//   NC SAF/Axes/Mover Axis 3 <-> TcCOM Objects/XtsProcessingUnit 1/Mover 3
//     SoftDrive 3/Data Pointer/InputPointer1 <-> Inputs/SoftDriveInput
//     SoftDrive 3/Data Pointer/OutputPointer1 <-> Outputs/SoftDriveOutput
//   NC SAF/Axes/Mover Axis 4 <-> TcCOM Objects/XtsProcessingUnit 1/Mover 4
//     SoftDrive 4/Data Pointer/InputPointer1 <-> Inputs/SoftDriveInput
//     SoftDrive 4/Data Pointer/OutputPointer1 <-> Outputs/SoftDriveOutput
//   NC SAF/Axes/Mover Axis 5 <-> TcCOM Objects/XtsProcessingUnit 1/Mover 5
//     SoftDrive 5/Data Pointer/InputPointer1 <-> Inputs/SoftDriveInput
//     SoftDrive 5/Data Pointer/OutputPointer1 <-> Outputs/SoftDriveOutput
//   NC SAF/Axes/Mover Axis 6 <-> TcCOM Objects/XtsProcessingUnit 1/Mover 6
//     SoftDrive 6/Data Pointer/InputPointer1 <-> Inputs/SoftDriveInput
//     SoftDrive 6/Data Pointer/OutputPointer1 <-> Outputs/SoftDriveOutput
//   NC SAF/Axes/Mover Axis 7 <-> TcCOM Objects/XtsProcessingUnit 1/Mover 7
//     SoftDrive 7/Data Pointer/InputPointer1 <-> Inputs/SoftDriveInput
//     SoftDrive 7/Data Pointer/OutputPointer1 <-> Outputs/SoftDriveOutput
//   NC SAF/Axes/Mover Axis 8 <-> TcCOM Objects/XtsProcessingUnit 1/Mover 8
//     SoftDrive 8/Data Pointer/InputPointer1 <-> Inputs/SoftDriveInput
//     SoftDrive 8/Data Pointer/OutputPointer1 <-> Outputs/SoftDriveOutput
//   NC SAF/Axes/Mover Axis 9 <-> TcCOM Objects/XtsProcessingUnit 1/Mover 9
//     SoftDrive 9/Data Pointer/InputPointer1 <-> Inputs/SoftDriveInput
//     SoftDrive 9/Data Pointer/OutputPointer1 <-> Outputs/SoftDriveOutput
//   Main Instance <-> NC SAF/Axes/Mover Axis 1
//     PlcTask Inputs/MAIN.Mover[0].AxisReference.NcToPlc <-> Outputs/ToPlc
//     PlcTask Outputs/MAIN.Mover[0].AxisReference.PlcToNc <-> Inputs/FromPlc
//   Main Instance <-> NC SAF/Axes/Mover Axis 10
//     PlcTask Inputs/MAIN.Mover[9].AxisReference.NcToPlc <-> Outputs/ToPlc
//     PlcTask Outputs/MAIN.Mover[9].AxisReference.PlcToNc <-> Inputs/FromPlc
//   Main Instance <-> NC SAF/Axes/Mover Axis 2
//     PlcTask Inputs/MAIN.Mover[1].AxisReference.NcToPlc <-> Outputs/ToPlc
//     PlcTask Outputs/MAIN.Mover[1].AxisReference.PlcToNc <-> Inputs/FromPlc
//   Main Instance <-> NC SAF/Axes/Mover Axis 3
//     PlcTask Inputs/MAIN.Mover[2].AxisReference.NcToPlc <-> Outputs/ToPlc
//     PlcTask Outputs/MAIN.Mover[2].AxisReference.PlcToNc <-> Inputs/FromPlc
//   Main Instance <-> NC SAF/Axes/Mover Axis 4
//     PlcTask Inputs/MAIN.Mover[3].AxisReference.NcToPlc <-> Outputs/ToPlc
//     PlcTask Outputs/MAIN.Mover[3].AxisReference.PlcToNc <-> Inputs/FromPlc
//   Main Instance <-> NC SAF/Axes/Mover Axis 5
//     PlcTask Inputs/MAIN.Mover[4].AxisReference.NcToPlc <-> Outputs/ToPlc
//     PlcTask Outputs/MAIN.Mover[4].AxisReference.PlcToNc <-> Inputs/FromPlc
//   Main Instance <-> NC SAF/Axes/Mover Axis 6
//     PlcTask Inputs/MAIN.Mover[5].AxisReference.NcToPlc <-> Outputs/ToPlc
//     PlcTask Outputs/MAIN.Mover[5].AxisReference.PlcToNc <-> Inputs/FromPlc
//   Main Instance <-> NC SAF/Axes/Mover Axis 7
//     PlcTask Inputs/MAIN.Mover[6].AxisReference.NcToPlc <-> Outputs/ToPlc
//     PlcTask Outputs/MAIN.Mover[6].AxisReference.PlcToNc <-> Inputs/FromPlc
//   Main Instance <-> NC SAF/Axes/Mover Axis 8
//     PlcTask Inputs/MAIN.Mover[7].AxisReference.NcToPlc <-> Outputs/ToPlc
//     PlcTask Outputs/MAIN.Mover[7].AxisReference.PlcToNc <-> Inputs/FromPlc
//   Main Instance <-> NC SAF/Axes/Mover Axis 9
//     PlcTask Inputs/MAIN.Mover[8].AxisReference.NcToPlc <-> Outputs/ToPlc
//     PlcTask Outputs/MAIN.Mover[8].AxisReference.PlcToNc <-> Inputs/FromPlc
//   Main Instance <-> NC SAF/Objects/Collision Avoidance
//     PlcTask Inputs/MAIN.GroupRef.NcToPlc <-> Group Outputs/ToPLC
//     PlcTask Outputs/MAIN.GroupRef.PlcToNc <-> Group Inputs/FromPLC

// ---- DUTs/HMI/HMIXTSHelper_typ.TcDUT
TYPE HMIXTSHelper_typ :
STRUCT
	Mover	: ARRAY[0..GVL.NUM_MOVERS-1] OF HMIXTSMoverHelper_typ;
END_STRUCT
END_TYPE

// ---- DUTs/HMI/HMIXTSMoverHelper_typ.TcDUT
TYPE HMIXTSMoverHelper_typ :
STRUCT
	BallImgVisibility:			BOOL;
	BallRejectImgVisibility:	BOOL;
	MoverTextVisibility: 		BOOL;
	MoverText: 					STRING;
END_STRUCT
END_TYPE

// ---- DUTs/IO/BallSeat/BallSeat_Inputs_typ.TcDUT
TYPE BallSeat_Inputs_typ:
STRUCT
	BallClampOpened AT %I*: BOOL;
	BallClampClosed AT %I*: BOOL;
	BallSeatExtended AT %I*: BOOL;
	BallSeatRetracted AT %I*: BOOL;
END_STRUCT
END_TYPE

// ---- DUTs/IO/BallSeat/BallSeat_Outputs_typ.TcDUT
TYPE BallSeat_Outputs_typ:
STRUCT
	BallClampOpen AT %Q*: BOOL;
	BallClampClose AT %Q*: BOOL;
	ExtendBallSeater AT %Q*: BOOL;
	RetractBallSeater AT %Q*: BOOL;
END_STRUCT
END_TYPE

// ---- DUTs/IO/Orient/Orient_IO_typ.TcDUT
TYPE Orient_IO_typ:
STRUCT
	Inputs	: Orient_Inputs_typ;
	Outputs	: Orient_Outputs_typ;
END_STRUCT
END_TYPE

// ---- DUTs/IO/Orient/Orient_Outputs_typ.TcDUT
TYPE Orient_Outputs_typ:
STRUCT
	BallClampOpen AT %Q*: BOOL;
	BallClampClose AT %Q*: BOOL;
	LoadBall AT %Q*: BOOL;
END_STRUCT
END_TYPE

// ---- DUTs/IO/IO_typ.TcDUT
TYPE IO_typ:
STRUCT
	Orient: 	Orient_IO_typ;
	BallSeat:	BallSeat_IO_typ;
	Print:		Print_IO_typ;
	Vision:		Vision_IO_typ;
	Kickout:	Kickout_IO_typ;
	TrayLoad:	TrayLoad_IO_typ;
END_STRUCT
END_TYPE

// ---- DUTs/IO/Print/Print_Inputs_typ.TcDUT
TYPE Print_Inputs_typ:
STRUCT
	PrintActive AT %I*: BOOL;
	PrintComplete AT %I*: BOOL;
END_STRUCT
END_TYPE

// ---- DUTs/IO/Print/Print_IO_typ.TcDUT
TYPE Print_IO_typ:
STRUCT
	Inputs	: Print_Inputs_typ;
	Outputs	: Print_Outputs_typ;
END_STRUCT
END_TYPE

// ---- DUTs/IO/Print/Print_Outputs_typ.TcDUT
TYPE Print_Outputs_typ:
STRUCT
	Print AT %Q*: BOOL;
END_STRUCT
END_TYPE

// ---- DUTs/IO/TrayLoad/TrayLoad_Inputs_typ.TcDUT
TYPE TrayLoad_Inputs_typ:
STRUCT
	BallClampOpened AT %I*: BOOL;
	BallClampClosed AT %I*: BOOL;
	TrayLoadComplete AT %I*: BOOL;
END_STRUCT
END_TYPE

// ---- DUTs/IO/TrayLoad/TrayLoad_IO_typ.TcDUT
TYPE TrayLoad_IO_typ:
STRUCT
	Inputs	: TrayLoad_Inputs_typ;
	Outputs	: TrayLoad_Outputs_typ;
END_STRUCT
END_TYPE

// ---- DUTs/IO/TrayLoad/TrayLoad_Outputs_typ.TcDUT
TYPE TrayLoad_Outputs_typ:
STRUCT
	BallClampOpen AT %Q*: BOOL;
	BallClampClose AT %Q*: BOOL;
	LoadTray AT %Q*: BOOL;
END_STRUCT
END_TYPE

// ---- DUTs/IO/Vision/Vision_Inputs_typ.TcDUT
TYPE Vision_Inputs_typ:
STRUCT
	VisionActive AT %I*: BOOL;
	VisionPass AT %I*: BOOL;
	VisionFail AT %I*: BOOL;
END_STRUCT
END_TYPE

// ---- DUTs/IO/Vision/Vision_IO_typ.TcDUT
TYPE Vision_IO_typ:
STRUCT
	Inputs	: Vision_Inputs_typ;
	Outputs	: Vision_Outputs_typ;
END_STRUCT
END_TYPE

// ---- POUs/XTS/BallPrinterStations/DUT/PrintConfig_typ.TcDUT
TYPE PrintConfig_typ :
STRUCT
	StationEnable	: ARRAY[0..GVL.MULTISTN_NUM_STN - 1] OF BOOL;
	ProcessIndex	: ARRAY[0..GVL.MULTISTN_NUM_STN - 1] OF USINT;
	FinalPrint		: ARRAY[0..GVL.MULTISTN_NUM_STN - 1] OF BOOL;
	LastProcessIndex0StnIndex	: USINT;
END_STRUCT
END_TYPE

// ---- POUs/XTS/BallPrinterStations/DUT/StnState_Enum.TcDUT
(*{attribute 'qualified_only'}*)
{attribute 'strict'}
TYPE StnState_Enum :
(
	STN_WAIT				:= 0,
	STN_CHECKMOVER			:= 1,
	STN_OPENBALLCLAMP		:= 2,
	STN_PROCESS				:= 3,
	STN_CLOSEBALLCLAMP		:= 4,
	STN_SEND				:= 5,
	STN_ERROR				:= 10
);
END_TYPE

// ---- GVLs/GVL.TcGVL
{attribute 'qualified_only'}
VAR_GLOBAL CONSTANT

    NUM_MOVERS   		: USINT := 10;   	// This should be set to the exact number of movers on the system
	NUM_ZONES			: USINT := 1;
    NUM_STATIONS 		: USINT := 5;   	// This should be set to a value equal to or greater than the number of stations needed
    NUM_MULTISTATIONS 	: USINT := 2;   	// This should be set to a value equal to or greater than the number of Multi stations needed
	MULTISTN_NUM_STN	: USINT := 4;		// This should be set to a value equal to or greater than the max number of stations in a multi station

    TRACK_LENGTH 		: LREAL := 3000;	// This should be set to the exact length [mm] of the track system

	STN_ORIENT		: USINT := 0;
	STN_BALLSEAT	: USINT := 1;
	STN_VISION		: USINT := 2;
	STN_KICKOUT		: USINT := 3;

	MULTISTN_PRINT		: USINT := 0;
	MULTISTN_TRAYLOAD	: USINT := 1;

    {attribute 'TcInitSymbol'}
    pXtsProcessingUnit : OTCID:=0; // This pointer needs to be initialized in the Main Instance, under Symbol Initialization

	NUM_TRACKS  : USINT := 1;	// This is the number of logical tracks in the system

END_VAR
VAR_GLOBAL
	newCallTime: LREAL;
END_VAR

// ---- ITFs/iMover.TcIO
INTERFACE iMover

METHOD ActivateTrack : BOOL
VAR_INPUT
	Track	: REFERENCE TO Track;
END_VAR
END_METHOD

{attribute 'monitoring' := 'call'}
PROPERTY CurrentDestinationPosition : LREAL
GET
END_GET
END_PROPERTY

{attribute 'monitoring' := 'call'}
PROPERTY CurrentMoveType : MoverCommandType_enum
GET
END_GET
END_PROPERTY

PROPERTY CurrentObjective : String
GET
END_GET
END_PROPERTY

PROPERTY CurrentTrack : POINTER TO Track
GET
END_GET
END_PROPERTY

METHOD Cyclic : iMover
VAR_IN_OUT
	GroupReference		: AXES_GROUP_REF;
END_VAR
END_METHOD

METHOD CyclicTrack : BOOL
VAR
END_VAR
END_METHOD

METHOD Disable : iMover
VAR_INPUT
END_VAR
END_METHOD

METHOD Enable : iMover
VAR_INPUT
END_VAR
END_METHOD

METHOD GroupStop : iMover
VAR_INPUT
END_VAR
END_METHOD

METHOD Halt : iMover
VAR_INPUT
END_VAR
END_METHOD

PROPERTY IsTrackReady : BOOL
GET
END_GET
END_PROPERTY

METHOD LogUserEvent : iMover
VAR_INPUT
	String1	: STRING;	// First content section of user-event message
	String2 : STRING;	// Second content section of user-event message
	String3 : STRING;	// Third content section of user-event message
END_VAR
END_METHOD

METHOD PUBLIC MoveToPosition : iMover
VAR_INPUT
	
	DestinationPosition		: LREAL;	// position on track for a shuttle to move towards

END_VAR
END_METHOD

METHOD MoveToStation : iMover
VAR_INPUT
	DestinationStation	: REFERENCE TO Station;	
END_VAR
END_METHOD

METHOD MoveVelocity : iMover
VAR_INPUT
	DesiredVelocity : LREAL;		//The velocity to be commanded [mm/s]
END_VAR
END_METHOD

PROPERTY Payload : Payload_typ
GET
END_GET
SET
END_SET
END_PROPERTY

METHOD ReissueCommand : iMover
VAR_INPUT
END_VAR
END_METHOD


METHOD SetAcceleration : iMover
VAR_INPUT
	Acceleration	: LREAL;
END_VAR
END_METHOD

METHOD SetDeceleration : iMover
VAR_INPUT
	Deceleration	: LREAL;
END_VAR
END_METHOD

METHOD SetDirection : iMover
VAR_INPUT
	Direction		: Tc3_Mc3Definitions.MC_Direction;
END_VAR
END_METHOD

METHOD SetJerk : iMover
VAR_INPUT
	Jerk		: LREAL;
END_VAR
END_METHOD

METHOD SetVelocity : iMover
VAR_INPUT
	Velocity		: LREAL;		// Updates Mover's internal velocity parameter. Takes effect immediately. [mm/s]
END_VAR
END_METHOD

METHOD SyncToAxis : iMover
VAR_INPUT
	
	MasterAxis		: REFERENCE TO AXIS_REF;
	MasterSyncPos	: LREAL;	// Master sync position (nonmodulo), where the input axis will be located when first synchronized
	SlaveSyncPos	: LREAL;	// Mover sync position, where the mover will be located when first synchronized
	SyncStrategy	: MC_SYNC_STRATEGY;	// Direction input
	
END_VAR
END_METHOD

METHOD SyncToMover : iMover
VAR_INPUT

	MasterMover		: REFERENCE TO Mover;	// Synchronization master mover, whose position to follow. Further motion commands break the pairing
	Gap				: LREAL;				// Gap distance to lead mover. Positive values indicate following, negative values indicate leading

END_VAR
END_METHOD

END_INTERFACE

// ---- POUs/XTS/Station.TcPOU
FUNCTION_BLOCK Station EXTENDS Objective
VAR

    {attribute 'hide'}
    internalPosition : LREAL;
	internalTrackId : DINT := 1;

END_VAR

{attribute 'monitoring' := 'variable'}
PROPERTY CurrentMover : REFERENCE TO Mover
GET
VAR

    i          : ULINT;
    difference : LREAL;

	moverTrackId: INT;
END_VAR
// default to unassigned
CurrentMover REF= 0;

FOR i := 0 TO SIZEOF(internalTrackedMovers) / SIZEOF(internalTrackedMovers[0]) - 1 DO

    // In order to deal with the rollover, we need to evaluate distance between congruence classes
    // e.g. On a 4m track, if the Station is at 0.34mm and the Mover is at 3999.8mm, then this is considered 'in position'	

    IF internalTrackedMovers[i] <> 0 THEN
		moverTrackId := internalTrackedMovers[i]^.CurrentTrack^.Id;
		IF (moverTrackId = internalTrackId) THEN

			difference := Position - internalTrackedMovers[i]^.TrackInfo.TrackPosition;
			// un-wrap if necessary
			IF (difference < 0) THEN 
				difference := difference + GVL.TRACK_LENGTH;
			END_IF
	
			IF (difference < 1.0) AND NOT internalTrackedMovers[i]^.Busy THEN
				CurrentMover                    REF= internalTrackedMovers[i]^;
				CurrentMover.SourceInstancePath := THIS^.InstancePath;
				// Exit;	// CW - shouldn't this be here?
			END_IF
		END_IF
    END_IF

END_FOR

// If the Station has no CurrentMover, then return an imposter ErrorMover, whose method calls all trigger an error message
IF __ISVALIDREF(CurrentMover) = FALSE THEN
    ErrorMover.SourceInstancePath := THIS^.InstancePath;
    CurrentMover                  REF= ErrorMover;
END_IF
END_GET
END_PROPERTY

METHOD Cyclic : BOOL

VAR
    i : USINT;
END_VAR
FOR i := 0 TO GVL.NUM_MOVERS - 1 DO

    // This mover is no longer destined for any station
    IF internalTrackedMovers[i] <> 0 AND_THEN internalTrackedMovers[i]^.CurrentMoveType <> MOVETYPE_STATION THEN
        internalTrackedMovers[i] := 0;
        // This mover is no longer destined for this specific station. Comparing instance path seems to be the best way to do this comparison?
    ELSIF internalTrackedMovers[i] <> 0 AND_THEN internalTrackedMovers[i]^.CurrentObjective <> InstancePath THEN
        internalTrackedMovers[i] := 0;
    END_IF

END_FOR
END_METHOD

{attribute 'monitoring' := 'variable'}
PROPERTY MoverInPosition : BOOL
GET
VAR

    i          : ULINT;
    difference : LREAL;
	moverTrackId: INT;
END_VAR
// default to false
MoverInPosition := FALSE;

FOR i := 0 TO SIZEOF(internalTrackedMovers) / SIZEOF(internalTrackedMovers[0]) - 1 DO

    // In order to deal with the rollover, we need to evaluate distance between congruence classes
    // e.g. On a 4m track, if the Station is at 0.34 mm and the Mover is at 3999.8mm, then this is considered 'in position' 

    // todo: make in-position tolerance adjustable. add condition that mover is stopped?
    IF internalTrackedMovers[i] <> 0 THEN
		moverTrackId := internalTrackedMovers[i]^.CurrentTrack^.Id;
		IF (moverTrackId = internalTrackId) THEN
			difference := Position - internalTrackedMovers[i]^.TrackInfo.TrackPosition;
			// un-wrap if necessary
			IF (difference < 0) THEN 
				difference := difference + GVL.TRACK_LENGTH;
			END_IF

			IF (difference < 1.0) AND NOT internalTrackedMovers[i]^.Busy THEN
				MoverInPosition := TRUE;
			END_IF
		END_IF;
    END_IF;

END_FOR
END_GET
END_PROPERTY

{attribute 'monitoring' := 'call'}
PROPERTY Position : LREAL
GET
Position := internalPosition;
END_GET
SET
internalPosition := Position;
END_SET
END_PROPERTY

PROPERTY TrackId : DINT
GET
TrackId := internalTrackId;
END_GET
SET
internalTrackId := TrackId;
END_SET
END_PROPERTY

END_FUNCTION_BLOCK

// ---- POUs/XTS/Objective.TcPOU
{attribute 'reflection'}
(*{attribute 'hide_all_locals'}*)
FUNCTION_BLOCK ABSTRACT Objective
VAR_INPUT
END_VAR
VAR

    internalTrackedMoverCount 	: USINT;
   
    internalTrackedMovers 		: ARRAY[0..GVL.NUM_MOVERS - 1] OF POINTER TO Mover;

    ErrorMover 					: ErrorMover;
	
    {attribute 'instance-path'}
    {attribute 'noinit'}
    InstancePath 				: STRING; // Unique variable path of the instance	
END_VAR
VAR_OUTPUT
END_VAR

PROPERTY CurrentMover : Reference to Mover
GET

// If no real mover can be returned as Current, return an imposter instead to output error messages
IF __ISVALIDREF( CurrentMover ) = FALSE THEN
	ErrorMover.SourceInstancePath	:= THIS^.InstancePath;
	CurrentMover					REF= ErrorMover;
END_IF
END_GET
END_PROPERTY

METHOD RegisterMover : BOOL
VAR_INPUT
    NewMover : REFERENCE TO Mover;
END_VAR

VAR
    i              : ULINT;
    duplicateFound : BOOL;
    emptyIDX       : ulint;
END_VAR
(*
	Add a mover to a list of movers tracked by the objective.
	Movers can't be added multiple times, so check for duplicates
	Movers can't overwrite others in the list, so check that the array element is clear
*)

IF __ISVALIDREF(NewMover) THEN // validate reference

    duplicateFound            := FALSE; // default to false, counterexample below
    internalTrackedMoverCount := 0;     // reset to zero, incremented below

    FOR i := 0 TO SIZEOF(internalTrackedMovers) / SIZEOF(internalTrackedMovers[i]) - 1 DO
        IF internalTrackedMovers[i] <> 0 THEN
            IF ADR(NewMover) = internalTrackedMovers[i] THEN
                duplicateFound := TRUE; // this mover already tracked
            END_IF

            internalTrackedMoverCount := internalTrackedMoverCount + 1;
        ELSE
            emptyIDX := i; // confirmed open array element
        END_IF
    END_FOR

    IF duplicateFound = FALSE THEN
        internalTrackedMovers[emptyIDX] := ADR(NewMover); // new mover goes into open array element
        internalTrackedMoverCount       := internalTrackedMoverCount + 1;
    END_IF

ELSE
    ADSLOGSTR(ADSLOG_MSGTYPE_LOG, 'Error: Mover input is invalid', '');
END_IF
END_METHOD

METHOD RegisterMoverList : BOOL
VAR_INPUT
    NewMoverList : iMoverList;
END_VAR
VAR
    i                : ULINT;
    duplicateFound   : BOOL;
    emptyIDX         : USINT;
    arrTrackedMovers : ARRAY[0..GVL.NUM_MOVERS - 1] OF POINTER TO Mover;
END_VAR
(*
	Adds an entire MoverList to the Tracked Movers of the objective.
*)

arrTrackedMovers := NewMoverList.TrackedMovers;

// IF __ISVALIDREF( NewMoverList ) THEN
IF NewMoverList <> 0 THEN
    FOR i := 0 TO SIZEOF(arrTrackedMovers) / SIZEOF(arrTrackedMovers[0]) - 1 DO

        THIS^.RegisterMover(arrTrackedMovers[i]^);

    END_FOR
END_IF
END_METHOD

{attribute 'monitoring' := 'call'}
PROPERTY TrackedMoverCount : USINT
GET
VAR
    i : INT;
END_VAR
TrackedMoverCount := 0;

FOR i := 0 TO GVL.NUM_MOVERS - 1 DO

    IF internalTrackedMovers[i] <> 0 THEN
        TrackedMoverCount := TrackedMoverCount + 1;
    END_IF

END_FOR
END_GET
END_PROPERTY

PROPERTY TrackedMovers : ARRAY[0..GVL.NUM_MOVERS - 1] OF POINTER TO Mover
GET
TrackedMovers := internalTrackedMovers;
END_GET
END_PROPERTY

METHOD UnregisterAll : BOOL
VAR_INPUT
END_VAR
VAR
    i : USINT;
END_VAR
// Blow out the tracked mover array
memset(ADR(internalTrackedMovers), 0, SIZEOF(internalTrackedMovers));
END_METHOD

METHOD UnregisterCurrent : BOOL
VAR_INPUT
END_VAR
THIS^.UnregisterMover(CurrentMover);
END_METHOD

METHOD UnregisterMover : BOOL
VAR_INPUT
    RemovingMover : REFERENCE TO Mover;
END_VAR
VAR
    i              : dint;
    duplicateFound : BOOL;
END_VAR
(*
	Remove a mover to a list of movers tracked by the objective.
	Only movers in the list can be removed, otherwise nothing happens
*)

//	IF RemovingMover <> 0 THEN			// validate pointer
IF __ISVALIDREF(RemovingMover) THEN

    internalTrackedMoverCount := 0;

    FOR i := 0 TO SIZEOF(internalTrackedMovers) / SIZEOF(internalTrackedMovers[0]) - 1 DO
        IF internalTrackedMovers[i] <> 0 THEN // validate pointer

            internalTrackedMoverCount := internalTrackedMoverCount + 1;

            IF ADR(RemovingMover) = internalTrackedMovers[i] THEN
                internalTrackedMovers[i]  := 0; // remove the pointer
                internalTrackedMoverCount := internalTrackedMoverCount - 1;
            END_IF

        END_IF
    END_FOR

ELSE
    ADSLOGSTR(ADSLOG_MSGTYPE_LOG, 'Error: Mover input is invalid', '');
END_IF
END_METHOD

END_FUNCTION_BLOCK

// ---- POUs/MAIN.TcPOU
PROGRAM MAIN
VAR
	// Machine Stations
	OrientStation:		OrientStation;
	BallSeatStation:	BallSeatStation;
	PrintStation:		PrintStation;
	VisionStation:		VisionStation;
	SimTimers:			SimTimers_typ;

	// ========= System Control / FSM Variables =========
	
	MainCommands 		: MainCommands_typ; 	// command struct for cycling thru the state machine
	MainState    		: MainState_enum;   	// enumeration for the Main state machine

	// ========= Linked NC Variables & References =========
	
	Mover    			: ARRAY[0..GVL.NUM_MOVERS - 1] OF Mover; 	// instantiation of Mover objects. Matches the number of movers on the system
    GroupRef 			: AXES_GROUP_REF;                       	 // linked to the Collision Avoidance group and passed cyclically to every Mover object

	// ========= Objectives & Parameters =========

    MoverList    		: MoverList;
    ParameterSet 		: MotionParameters_typ;

    Station         	: ARRAY[0..GVL.NUM_STATIONS - 1] OF Station;
	MultiStation		: ARRAY[0..GVL.NUM_MULTISTATIONS - 1] OF MultiStation;
    Zone            	: ARRAY[0..0] OF Zone;

    // ========= Example Application Variables =========

    lowVelocity    		: LREAL := 200;  	// mm/s
    mediumVelocity 		: LREAL := 800;  	// mm/s
    highVelocity   		: LREAL := 1200; 	// mm/s

    // ========= Helper, State, & Index Variables =========
	
    i                	: UINT; 	// index variable; gets reused in various FOR loops
	j					: UINT;		// index variable; gets reused in various FOR loops
    n                	: UINT; 	// secondary index variable, for enabling movers
    allMoversEnabled 	: BOOL; 	// helper flag for verifying enable status of all movers
	allMoverTracksEnabled : BOOL;	// helper flag for verifying track active status of all movers
	allMoversDisabled	: BOOL;		// helper flag for verifying disable status of all movers
	allMoversHalted		: BOOL;		// helper flag for verifying halt status of all movers

    StationTimer 		: ARRAY[0..GVL.NUM_STATIONS-1] OF TON; // timer blocks, for station dwells	
    MultiStationTimer 	: ARRAY[0..GVL.NUM_MultiSTATIONS-1] OF TON; // timer blocks, for station dwells	
	
	// ========= XTS Utility Diagnostics =========
	
	VisuDiag						: FB_VisuXtsDiag;
	fbXtsEnvironment				: FB_TcIoXtsEnvironment;
	fbXtsEnvironmentVisu			: FB_XtsEnvironmentVisu;
	stXtsEnvironmentConfiguration	: ST_XtsEnvironmentConfiguration;
	nEnvironmentState				: INT;
	
	// ======== Track management ========
	Track		: ARRAY [0..GVL.NUM_TRACKS] OF Track;

	// IO
	IO: IO_typ;

	Payload: Payload_typ;
	HMIXTSHelper : HMIXTSHelper_typ;
END_VAR

(* ======================================================================================

--- XTS Starter Project ---

This MAIN (PRG) is intended to serve as an example, which can be modified to suit your specific application.

No programming changes should be necessary inside the provided XTS objects / function block definitions.
They are intended to be simply instantiated and controlled via the provided methods and properties.
However the objects are provided as open-source for modification and extension as needed.

Documentation for these objects can be found online at:
https://beckhoff-usa-community.github.io/XTS_Base/

Bug reports, new feature requests, and general feedback is always welcome on our Github page.
For any other questions, please reach out to your local Application Engineer.

- Beckhoff USA Advanced Applications Group

====================================================================================== *)
_AppInfo.KeepOutputsOnBP := TRUE;
CASE MainState OF
    MS_DISABLED: // --------------------------------------------------------- IDLE STATE
		(*Wait here until an operator issues a MainCommand to Enable the system. 
		Disallow Start and Stop commands until the system has been Enabled*)

        MainCommands.Start		:= FALSE;
		MainCommands.Stop		:= FALSE;
		
        IF MainCommands.Enable THEN
            MainCommands.Disable := FALSE;
            MainState            := MS_INITIALIZING_MOVERS;
        END_IF

    MS_INITIALIZING_MOVERS: // --------------------------------------------- SET MOVER MOTION PARAMETERS
		(*Initialize Mover motion parameters via a Parameter Set. Once complete, step
		forward to begin Enabling movers on the system*)
		
		ParameterSet.Jerk         := 1E5; // mm/s3
		ParameterSet.Acceleration := 1E4; // mm/s2
		ParameterSet.Deceleration := 1E4; // mm/s2
		ParameterSet.Velocity     := 1E3; // mm/s
		ParameterSet.Direction    := mcDirectionPositive;

        FOR i := 0 TO GVL.NUM_MOVERS - 1 DO
            Mover[i].MotionParameters := ParameterSet;
        END_FOR
		
		IF MainCommands.Disable THEN
			MainCommands.Enable		:= FALSE;
			MainState				:= MS_DISABLED;
		ELSIF MainCommands.Stop THEN
			MainCommands.Stop		:= FALSE;
			MainCommands.Disable	:= TRUE;
			MainCommands.Start		:= FALSE;
			MainState				:= MS_DISABLED;
		ELSIF MainCommands.Enable THEN
        	MainState 				:= MS_ONESHOT_ENABLE;
		END_IF

	MS_ONESHOT_ENABLE:	// -------------------------------------------------- SINGLE-CYCLE ISSUE ENABLE COMMANDS
		(*Begin Enabling movers by calling Mover.Enable(). Methods in this project
		are intended to be called once, although they will function correctly if called repeatedly*)

		FOR i := 0 TO GVL.NUM_MOVERS - 1 DO
			Mover[i].Enable();
		END_FOR

		MainState		:= MS_ENABLING_MOVERS;
	
    MS_ENABLING_MOVERS: // -------------------------------------------------- RESETTING AND ENABLING AXES
		(*Wait here until all movers have Enabled. This means that the Axis has
		fully energized, and also that all Collision Avoidance grouping and Mover 1 detection
		has finished. If the state machine gets stuck in this state, check the Error output
		of an individual Mover to see what the issue is. A common cause is forgetting to link
		Mover NC Axes to the AXIS_REF inside the PLC*)

        allMoversEnabled := TRUE; // default ...

        FOR i := 0 TO GVL.NUM_MOVERS - 1 DO
            IF Mover[i].Ready = FALSE THEN
                allMoversEnabled 		:= FALSE;
            END_IF
        END_FOR

        IF allMoversEnabled THEN
			IF MainCommands.Disable THEN
				MainCommands.Enable		:=FALSE;
            	MainState				:= MS_ONESHOT_DISABLE;
			ELSIF MainCommands.Stop	 THEN
				MainCommands.Start		:=FALSE;
				MainState				:= MS_ONESHOT_STOP;
			ELSIF MainCommands.Enable THEN
	        	MainState 				:= MS_INITIALIZING_OBJECTIVES;
			END_IF
        END_IF

    MS_INITIALIZING_OBJECTIVES: // --------------------------------------------- WRITING OBJECTIVE PARAMETERS
		(*Initialize Station positions, Position Trigger positions, Zones etc. *)

        // Initialize station positions
        Station[GVL.STN_ORIENT].Position	:= 800;
        Station[GVL.STN_BALLSEAT].Position	:= 900;
        Station[GVL.STN_VISION].Position	:= 2125;
        Station[GVL.STN_KICKOUT].Position	:= 2375;

		MultiStation[GVL.MULTISTN_PRINT].PositionTrigger.Position	:= 1541;
		MultiStation[GVL.MULTISTN_PRINT].Station[0].Position		:= 1621;
		MultiStation[GVL.MULTISTN_PRINT].Station[1].Position		:= 1707;
		MultiStation[GVL.MULTISTN_PRINT].Station[2].Position		:= 1793;
		MultiStation[GVL.MULTISTN_PRINT].Station[3].Position		:= 1879;

		MultiStation[GVL.MULTISTN_TRAYLOAD].PositionTrigger.Position	:= 41;
		MultiStation[GVL.MULTISTN_TRAYLOAD].Station[0].Position			:= 121;
		MultiStation[GVL.MULTISTN_TRAYLOAD].Station[1].Position			:= 207;
		MultiStation[GVL.MULTISTN_TRAYLOAD].Station[2].Position			:= 293;
		MultiStation[GVL.MULTISTN_TRAYLOAD].Station[3].Position			:= 379;

        Zone[0].StartPosition := 0;
        Zone[0].EndPosition   := 3000;

		// give all tracks their ID number
		FOR i := 0 TO GVL.NUM_TRACKS DO
			Track[i].Id := UINT_TO_INT(i);
		END_FOR
		
		// If a single logical track is used (typically aa closed loop) then tracks to not need to be initialized
		Track[0].OTCID := 0;				// special "absolute reference" case for a single closed loop
		Track[1].OTCID:= 16#010100C0;		// value copied from XtsProcessingUnit1 > Track x > Object > Object Id field

		MainState := MS_ACTIVATE_TRACKS;
		
	MS_ACTIVATE_TRACKS:
		// activate all movers on track[0]
		FOR i := 0 TO GVL.NUM_MOVERS - 1 DO
            Mover[i].ActivateTrack(Track[1]);
        END_FOR
		
		MainState := MS_WAIT_FOR_TRACKS;
	
	MS_WAIT_FOR_TRACKS:
		// wait for all movers to activate their tracks
		
		allMoverTracksEnabled := TRUE;
		FOR i := 0 TO GVL.NUM_MOVERS - 1 DO
			IF (NOT Mover[i].IsTrackReady) THEN
            	allMoverTracksEnabled := FALSE;
			END_IF;
        END_FOR
		IF (allMoverTracksEnabled) THEN
			MainState := MS_ENABLED;	
		END_IF

    MS_ENABLED: // ------------------------------------------------------------- MOVERS ENABLED, STOPPED
		(*In this state, Movers should be energized and holding their position. They should wait
		until a Start command is issued. This is also a good state to include basic Recovery steps.
		Our example shows a simple use-case involving Zones for localized recovery*)

		MainCommands.Stop	:= FALSE;
	
        IF MainCommands.Start THEN

            // ===== RECOVERY LOGIC =====

            (*
			Recovery is typically very application-specific. Each implementation will need to determine
			what to do with work-in-progres, rejects, movers with unknown product status, etc.s
			*)

            // Register all movers with all Zones, for recovery
            FOR i := 0 TO GVL.NUM_MOVERS - 1 DO
				FOR j := 0 TO GVL.NUM_ZONES - 1 DO
					Zone[j].RegisterMover( Mover[i] );
				END_FOR
            END_FOR
			
            Zone[0].CurrentMoverList.SetAllVelocity(1500).MoveAllToStation(Station[GVL.STN_ORIENT]);

            // ===== END =====

            MainState			:= MS_RUN;

        ELSIF MainCommands.Disable THEN
            MainCommands.Enable := FALSE;
            MainState           := MS_ONESHOT_STOP;
        END_IF

    MS_RUN: // --------------------------------------------------------------- OPERATING
		(*Mover routing logic should be written here to define the system's operating behavior.
		Station implementations, Position Trigger logic, etc. In general, you can remove the example code
		here down to the short line break that looks like this: // ============= *)

		OrientStation.Run	:= TRUE;
		BallSeatStation.Run	:= TRUE;
		PrintStation.Run	:= TRUE;
		VisionStation.Run	:= TRUE;
	
        // Vision Station Logic	
		// Station specific logic to be moved to FUB
//        IF Station[GVL.STN_VISION].MoverInPosition THEN
//            StationTimer[GVL.STN_VISION](IN := TRUE, PT := T#250MS);
//            IF StationTimer[GVL.STN_VISION].Q THEN
//                Station[GVL.STN_VISION].CurrentMover.MoveToStation(Station[GVL.STN_ORIENT]);
//            END_IF
//        ELSE
//            StationTimer[GVL.STN_VISION](IN := FALSE);
//        END_IF

		// Kickout Station Logic
		// Station specific logic to be moved to FUB
        IF Station[GVL.STN_KICKOUT].MoverInPosition THEN
            StationTimer[GVL.STN_KICKOUT](IN := TRUE, PT := T#1000MS);
            IF StationTimer[GVL.STN_KICKOUT].Q THEN
				// maybe write a function to remove all ball data when ball is removed?
				Payload				:= Station[GVL.STN_KICKOUT].CurrentMover.Payload;
				Payload.HasBall		:= FALSE;	
				Payload.Reject		:= FALSE;
				Payload.BallSeated	:= FALSE;
				Station[GVL.STN_KICKOUT].CurrentMover.Payload	:= Payload;
                Station[GVL.STN_KICKOUT].CurrentMover.MoveToStation(Station[GVL.STN_ORIENT]);
            END_IF
        ELSE
            StationTimer[GVL.STN_KICKOUT](IN := FALSE);
        END_IF

		// Tray Load Station Logic
		IF MultiStation[GVL.MULTISTN_TRAYLOAD].Station[0].MoverInPosition THEN
			MultiStationTimer[GVL.MULTISTN_TRAYLOAD](IN := TRUE, PT := T#1500MS);
			IF MultiStationTimer[GVL.MULTISTN_TRAYLOAD].Q THEN
				FOR i := 0 TO 3 DO
					MultiStation[GVL.MULTISTN_TRAYLOAD].Station[i].CurrentMover.MoveToStation(Station[GVL.STN_ORIENT]);
				END_FOR
				MultiStationTimer[GVL.MULTISTN_TRAYLOAD](IN := FALSE);
			END_IF
		ELSE
			MultiStationTimer[GVL.MULTISTN_TRAYLOAD](IN := FALSE);
		END_IF

		// Example call to XTS Utility library. See Diagnostics section of docs for more info
		(*
		myMoverMileage	:= fbXtsEnvironment.XpuTcIo(1).MoverTcIo(2).GetDistanceDriven();
		*)
		
		// =============

        IF MainCommands.Stop THEN
            MainCommands.Start 	:= FALSE;
            MainState         	:= MS_ONESHOT_STOP;
        ELSIF MainCommands.Disable THEN
            MainCommands.Enable := FALSE;
            MainState           := MS_ONESHOT_STOP;
        END_IF
		
	MS_ONESHOT_STOP:	// --------------------------------------------------- SINGLE-CYCLE ISSUE HALT COMMANDS
		(*Issue a halt command, then change states right away to wait for Movers to carry out the instruction*)
	
		FOR i := 0 TO GVL.NUM_MOVERS - 1 DO
			Mover[i].Halt();
		END_FOR

		OrientStation.Run	:= FALSE;
		BallSeatStation.Run	:= FALSE;
		PrintStation.Run	:= FALSE;
	
		MainState					:= MS_STOPPING;
	
    MS_STOPPING: // ---------------------------------------------------------- STOPPING MOVERS
		(*Movers are coming to a stop here in this state*)

		// Stop all movers
		allMoversHalted				:= TRUE;
		FOR i := 0 TO GVL.NUM_MOVERS - 1 DO
			Mover[i].AxisReference.ReadStatus();
			IF Mover[i].AxisReference.Status.Moving THEN
				allMoversHalted		:= FALSE;
			END_IF
		END_FOR
		
		MainCommands.Start			:= FALSE;
 
		IF allMoversHalted THEN
           	MainState 				:= MS_STOPPED;
		END_IF
        

    MS_STOPPED: // ------------------------------------------------------------ Stop Command has been sent, hold here
		(*Movers are now stopped, and further Main Commands can be issued to the system*)

        IF MainCommands.Disable THEN
            MainCommands.Enable 	:= FALSE;
			MainCommands.Start		:= FALSE;
            MainState           	:= MS_ONESHOT_DISABLE;
        ELSIF MainCommands.Start THEN
            MainCommands.Stop 		:= FALSE;
            MainState         		:= MS_ENABLING_MOVERS;
        END_IF

        // Unregister everything from all stations
        FOR i := 0 TO GVL.NUM_STATIONS - 1 DO
            Station[i].UnregisterAll();
        END_FOR

        // Unregister everything from all stations
        FOR i := 0 TO GVL.NUM_MULTISTATIONS - 1 DO
            MultiStation[i].UnregisterAll();
        END_FOR

//        // Unregister everything from all Pos Trigs
//        FOR i := 0 TO SIZEOF(PositionTrigger) / SIZEOF(PositionTrigger[0]) - 1 DO
//            PositionTrigger[i].UnregisterAll();
//        END_FOR

//        // Unregister everything from all speed trigs
//        FOR i := 0 TO SIZEOF(SpeedTrigger) / SIZEOF(SpeedTrigger[0]) - 1 DO
//            SpeedTrigger[i].UnregisterAll();
//        END_FOR

        // Unregister everything from all zones
        FOR i := 0 TO SIZEOF(Zone) / SIZEOF(Zone[0]) - 1 DO
            Zone[i].UnregisterAll();
        END_FOR
	
	MS_ONESHOT_DISABLE:	// ------------------------------------------------------- SINGLE CYCLE ISSUE DISABLE COMMANDS
		(*Mover disable commands are issued here, followed by a state tranisition to await completion of the Disabling*)
		FOR i := 0 TO GVL.NUM_MOVERS DO
			Mover[i].Disable();
		END_FOR

		MainState					:=	MS_DISABLING;
	
    MS_DISABLING: // --------------------------------------------------- DISABLING MOVERS
		(*Movers are Disabling. During this step, we also Unregister movers from relevant Objectives
		to ensure proper startup behavior*)

        // Unregister everything from all stations
        FOR i := 0 TO GVL.NUM_STATIONS - 1 DO
            Station[i].UnregisterAll();
        END_FOR

		// Unregister everything from all multi stations
		FOR i := 0 TO GVL.NUM_MULTISTATIONS - 1 DO
			MultiStation[i].UnregisterAll();
		END_FOR

//        // Unregister everything from all Position triggers
//        FOR i := 0 TO SIZEOF(PositionTrigger) / SIZEOF(PositionTrigger[0]) - 1 DO
//            PositionTrigger[i].UnregisterAll();
//        END_FOR

//        // Unregister everything from all speed triggers
//        FOR i := 0 TO SIZEOF(SpeedTrigger) / SIZEOF(SpeedTrigger[0]) - 1 DO
//            SpeedTrigger[i].UnregisterAll();
//        END_FOR

        // Unregister everything from all zones
        FOR i := 0 TO SIZEOF(Zone) / SIZEOF(Zone[0]) - 1 DO
            Zone[i].UnregisterAll();
        END_FOR
		
		allMoversDisabled				:= TRUE;
		
		FOR i := 0 TO gvl.NUM_MOVERS-1 DO
			IF NOT Mover[i].AxisReference.Status.Disabled THEN 
				allMoversDisabled		:= FALSE;
			END_IF
		END_FOR
 
        IF allMoversDisabled THEN
            MainState					:= MS_DISABLED;
        END_IF

    MS_ERROR: // --------------------------------------------------- ERRORSTATE
		(*A reset command can be included here to clear Mover errors, etc. and return
		to a controlled state*)

    MS_DEBUG: // ------------------------------------------------------- DEV USE ONLY
		(*This state is intentionally left blank, 
		for optional use by a developer during programming*)

END_CASE;

// Station Actions
ACT_Orient();
ACT_BallSeat();
ACT_Print();
ACT_Vision();
ACT_IOSim();

ACT_HMIHelper();

// Initialize and update diagnostic features
InitializeUtilityLibrary();

// Call all mover function blocks cyclically
FOR i := 0 TO GVL.NUM_MOVERS - 1 DO
    Mover[i].Cyclic(GroupRef);
	Mover[i].AxisReference.ReadStatus();
END_FOR;

// Call all station function blocks cyclically
FOR i := 0 TO GVL.NUM_STATIONS - 1 DO
    Station[i].Cyclic();
END_FOR

FOR i := 0 TO GVL.NUM_MULTISTATIONS - 1 DO
	MultiStation[i].Cyclic();
END_FOR

ACTION ACT_BallSeat:
// INIT
BallSeatStation.rStation		REF= Station[GVL.STN_BALLSEAT];
BallSeatStation.rIO				REF= IO.BallSeat;
BallSeatStation.rPrintStation	REF= MultiStation[GVL.MULTISTN_PRINT];

// Inputs
BallSeatStation.Enable	:= MainCommands.Enable;

// FB CALLS
BallSeatStation();
END_ACTION

ACTION ACT_HMIHelper:
FOR i := 0 TO gvl.NUM_MOVERS - 1 DO
	Payload	:= Mover[i].Payload;
	HMIXTSHelper.Mover[i].BallImgVisibility			:= Payload.HasBall AND NOT Payload.Reject;
	HMIXTSHelper.Mover[i].BallRejectImgVisibility	:= Payload.HasBall AND Payload.Reject;
	HMIXTSHelper.Mover[i].MoverTextVisibility		:= Payload.HasBall;
	CASE Payload.PlayerNumber OF
	1:		HMIXTSHelper.Mover[i].MoverText		:= '1';
	2:		HMIXTSHelper.Mover[i].MoverText		:= '2';
	3:		HMIXTSHelper.Mover[i].MoverText		:= '3';
	4:		HMIXTSHelper.Mover[i].MoverText		:= '4';
	ELSE	HMIXTSHelper.Mover[i].MoverText		:= 'InvalidText';
	END_CASE
END_FOR
END_ACTION

ACTION ACT_IOSim:
// Orient
SimTimers.TON_Orient_OpenBallClamp(IN := IO.Orient.Outputs.BallClampOpen AND NOT IO.Orient.Outputs.BallClampClose, PT := T#150MS);
SimTimers.TON_Orient_CloseBallClamp(IN := IO.Orient.Outputs.BallClampClose AND NOT IO.Orient.Outputs.BallClampOpen, PT := T#150MS);
SimTimers.TON_Orient_LoadBall(IN := IO.Orient.Outputs.LoadBall, PT := T#700MS);

IF SimTimers.TON_Orient_CloseBallClamp.Q THEN		IO.Orient.Inputs.BallClampClosed	:= TRUE;	IO.Orient.Inputs.BallClampOpened	:= FALSE;	END_IF
IF SimTimers.TON_Orient_OpenBallClamp.Q THEN		IO.Orient.Inputs.BallClampOpened	:= TRUE;	IO.Orient.Inputs.BallClampClosed	:= FALSE;	END_IF
IO.Orient.Inputs.BallLoadComplete					:= SimTimers.TON_Orient_LoadBall.Q;

// Ball Seater
SimTimers.TON_BallSeat_OpenBallClamp(IN := IO.BallSeat.Outputs.BallClampOpen AND NOT IO.BallSeat.Outputs.BallClampClose, PT := T#150MS);
SimTimers.TON_BallSeat_CloseBallClamp(IN := IO.BallSeat.Outputs.BallClampClose AND NOT IO.BallSeat.Outputs.BallClampOpen, PT := T#150MS);
SimTimers.TON_BallSeat_ExtendBallSeater(IN := IO.BallSeat.Outputs.ExtendBallSeater AND NOT IO.BallSeat.Outputs.RetractBallSeater, PT := T#150MS);
SimTimers.TON_BallSeat_RetractBallSeater(IN := IO.BallSeat.Outputs.RetractBallSeater AND NOT IO.BallSeat.Outputs.ExtendBallSeater, PT := T#150MS);

IF SimTimers.TON_BallSeat_CloseBallClamp.Q THEN		IO.BallSeat.Inputs.BallClampClosed		:= TRUE;	IO.BallSeat.Inputs.BallClampOpened		:= FALSE;	END_IF
IF SimTimers.TON_BallSeat_OpenBallClamp.Q THEN		IO.BallSeat.Inputs.BallClampOpened		:= TRUE;	IO.BallSeat.Inputs.BallClampClosed		:= FALSE;	END_IF
IF SimTimers.TON_BallSeat_ExtendBallSeater.Q THEN	IO.BallSeat.Inputs.BallSeatExtended		:= TRUE;	IO.BallSeat.Inputs.BallSeatRetracted	:= FALSE;	END_IF
IF SimTimers.TON_BallSeat_RetractBallSeater.Q THEN	IO.BallSeat.Inputs.BallSeatRetracted	:= TRUE;	IO.BallSeat.Inputs.BallSeatExtended		:= FALSE;	END_IF

// Printer
SimTimers.TON_Print_PrintComplete(IN := IO.Print.Outputs.Print, PT := T#1200MS);

IO.Print.Inputs.PrintActive		:= SimTimers.TON_Print_PrintComplete.IN AND NOT SimTimers.TON_Print_PrintComplete.Q;
IO.Print.Inputs.PrintComplete	:= SimTimers.TON_Print_PrintComplete.Q;

// Vision
SimTimers.TON_Vision_ScanBall(IN := IO.Vision.Outputs.Inspect, PT := T#1000MS);
IO.Vision.Inputs.VisionActive := IO.Vision.Outputs.Inspect AND NOT(SimTimers.TON_Vision_ScanBall.Q);
IF SimTimers.TON_Vision_ScanBall.Q THEN	IO.Vision.Inputs.VisionPass	:= FALSE;	IO.Vision.Inputs.VisionFail	:= TRUE;
ELSE IO.Vision.Inputs.VisionPass	:= FALSE;	IO.Vision.Inputs.VisionFail	:= FALSE;	END_IF;
END_ACTION

ACTION ACT_Orient:
// INIT
OrientStation.rStation		REF= Station[GVL.STN_ORIENT];
OrientStation.rIO			REF= IO.Orient;
OrientStation.rBallSeatStn	REF= Station[GVL.STN_BALLSEAT];
OrientStation.rKickoutStn	REF= Station[GVL.STN_KICKOUT];

// Inputs
OrientStation.Enable	:= MainCommands.Enable;

// FB CALLS
OrientStation();
END_ACTION

ACTION ACT_Print:
// INIT
PrintStation.rMultiStn			REF= MultiStation[GVL.MULTISTN_PRINT];
PrintStation.rIO				REF= IO.Print;
PrintStation.rVisionStation		REF= Station[GVL.STN_VISION];
PrintStation.rKickoutStation	REF= Station[GVL.STN_KICKOUT];

// Inputs
PrintStation.Enable		:= MainCommands.Enable;
PrintStation.NumColor	:= 2;
PrintStation.NumIndex	:= 2;

// FB CALLS
PrintStation();
END_ACTION

ACTION ACT_Vision:
// INIT
VisionStation.rStation			REF= Station[GVL.STN_VISION];
VisionStation.rIO				REF= IO.Vision;
VisionStation.rKickoutStation	REF= Station[GVL.STN_KICKOUT];
VisionStation.rTrayloadStation	REF= Station[GVL.MULTISTN_TRAYLOAD];

// Inputs
VisionStation.Enable	:= MainCommands.Enable;

// FB CALLS
VisionStation();
END_ACTION

ACTION InitializeUtilityLibrary:



CASE nEnvironmentState OF
	0:	// ----------------------------------------- Enable Init Items
	
		// Enable init Info Server if needed
		stXtsEnvironmentConfiguration.bEnableInitInfoServer		:= TRUE;
		
		// Enable init CA Group if needed
		stXtsEnvironmentConfiguration.bEnableInitCaGroup		:= TRUE;
		
		// Set configuration of XtsUtility init
		fbXtsEnvironment.P_XtsEnvironmentConfiguration			:= stXtsEnvironmentConfiguration;
		
		// Next step
		nEnvironmentState	:= 1;
		
	1:	// ------------------------------------------ Init Environment
		
		// Start init
		IF fbXtsEnvironment.Init(TRUE) THEN
			// stop init
			fbXtsEnvironment.Init(FALSE);
			
			// next step
			nEnvironmentState	:= 2;
		END_IF
		
	2:	// ------------------------------------------ Check for success
	
		// Check IsInitialized property
		IF fbXtsEnvironment.P_IsInitialized THEN
			// next step
			nEnvironmentState	:= 3;
		END_IF
		
	3:	// ------------------------------------------- Init Visu
	
		fbXtsEnvironmentVisu( ipTcIoXtsEnvironment := fbXtsEnvironment );
		
		// next step
		nEnvironmentState	:= 4;
		
	4:	// ------------------------------------------- Init done

		fbXtsEnvironmentVisu.Cycle();
		
END_CASE
END_ACTION

END_PROGRAM

// ---- POUs/XTS/BallPrinterStations/BallSeatStation.TcPOU
FUNCTION_BLOCK BallSeatStation EXTENDS MachineStation
VAR_INPUT
	rIO				: REFERENCE TO BallSeat_IO_typ;
	rStation		: REFERENCE TO Station;
	rPrintStation	: REFERENCE TO MultiStation;
END_VAR
VAR_OUTPUT
END_VAR
VAR
	test:INT;
	Payload	: Payload_typ;
END_VAR

IF NOT (__ISVALIDREF(rStation) AND __ISVALIDREF(rIO) AND __ISVALIDREF(rPrintStation)) THEN
	ADSLOGSTR( ADSLOG_MSGTYPE_ERROR, 'Invalid reference at %s.', InstancePath);	// how to make this work?
	RETURN;
END_IF

// WHATS THE DIFFERENCE BETWEEN PUTTING THIS HERE VS FB.Cyclic Method?

IF Enable THEN
	IF NOT _Enable THEN
		;
	END_IF

	CASE State OF
		STN_WAIT:
			IF Run AND rStation.MoverInPosition THEN
				Payload						:= rStation.CurrentMover.Payload;
				rIO.Outputs.BallClampOpen	:= TRUE;
				State						:= STN_OPENBALLCLAMP;
			END_IF

		STN_OPENBALLCLAMP:
			IF rIO.Inputs.BallClampOpened THEN
				rIO.Outputs.BallClampOpen		:= FALSE;
				rIO.Outputs.ExtendBallSeater	:= TRUE;
				State							:= STN_PROCESS;
			END_IF

		STN_PROCESS:
			IF rIO.Inputs.BallSeatExtended THEN
				rIO.Outputs.ExtendBallSeater	:= FALSE;
				rIO.Outputs.RetractBallSeater	:= TRUE;
				Payload.BallSeated				:= TRUE;
				rIO.Outputs.BallClampClose		:= TRUE;
				State							:= STN_CLOSEBALLCLAMP;
			END_IF

		STN_CLOSEBALLCLAMP:
			IF rIO.Inputs.BallClampClosed AND rIO.Inputs.BallSeatRetracted THEN
				rIO.Outputs.RetractBallSeater	:= FALSE;
				rIO.Outputs.BallClampClose		:= FALSE;
				State							:= STN_SEND;
			END_IF

		STN_SEND:
			IF Test = 7 THEN Payload.Reject	:= TRUE; END_IF	// TEMP - TO TEST PRINT STATION REJECT HANDLING
			Test := SEL(Test >= 7, Test + 1, 0);	

			rStation.CurrentMover.Payload	:= Payload;
			rStation.CurrentMover.MoveToMultiStation(rPrintStation);
			rStation.UnregisterCurrent();
			State							:= STN_WAIT;
		
		STN_ERROR:
	
	END_CASE

ELSIF _Enable THEN
	rIO.Outputs.BallClampClose		:= FALSE;
	rIO.Outputs.BallClampOpen		:= FALSE;
	rIO.Outputs.ExtendBallSeater	:= FALSE;
	rIO.Outputs.RetractBallSeater	:= FALSE;
	State	:= STN_WAIT;
END_IF

//Save Previous Values
_Enable	:= Enable;

END_FUNCTION_BLOCK

// ---- POUs/XTS/MultiStation.TcPOU
FUNCTION_BLOCK MultiStation(* EXTENDS Objective*);
VAR_INPUT
	PositionTrigger		: PositionTrigger;
	Station				: ARRAY[0..GVL.MULTISTN_NUM_STN - 1] OF Station;
END_VAR
VAR_OUTPUT
END_VAR
VAR
	i: INT;
    internalTrackedMoverCount 	: USINT;
	
    {attribute 'hide'}
    internalPosition : LREAL;
	internalTrackId : DINT; 

    {attribute 'instance-path'}
    {attribute 'noinit'}
    InstancePath 				: STRING; // Unique variable path of the instance
END_VAR

{attribute 'monitoring' := 'variable'}
PROPERTY AllMoversInPosition : BOOL
GET
VAR

    i          : ULINT;
	TrackedMovers	: UINT;
END_VAR
// default to false
AllMoversInPosition := TRUE;
TrackedMovers		:= 0;

FOR i := 0 TO SIZEOF(Station) / SIZEOF(Station[0]) - 1 DO
	IF Station[i].TrackedMoverCount > 0 THEN
		TrackedMovers	:= TrackedMovers + 1;
		IF NOT Station[i].MoverInPosition THEN
			AllMoversInPosition	:= FALSE;
			EXIT;
		END_IF
	END_IF
END_FOR

IF TrackedMovers = 0 THEN
	AllMoversInPosition	:= FALSE;
END_IF
END_GET
END_PROPERTY

METHOD Cyclic : BOOL
VAR
	i : USINT;
END_VAR
//IF PositionTrigger.MoverPassedPosition THEN
//	PositionTrigger.CurrentMover.MoveToStation(Station[0]);
//	PositionTrigger.MuteCurrent();
//END_IF

// Call Cyclics
PositionTrigger.Cyclic();
FOR i := 0 TO GVL.MULTISTN_NUM_STN - 1 DO
	Station[i].Cyclic();
END_FOR
END_METHOD

{attribute 'monitoring' := 'call'}
PROPERTY Position : LREAL
GET
InternalPosition	:= Station[0].Position;
Position 			:= internalPosition;
Position;
END_GET
END_PROPERTY

METHOD RegisterMover : BOOL
VAR_INPUT
    NewMover : REFERENCE TO Mover;
END_VAR
(*
	Add a mover to a list of movers tracked by the objective.
	Movers can't be added multiple times, so check for duplicates
	Movers can't overwrite others in the list, so check that the array element is clear
*)
PositionTrigger.RegisterMover(NewMover);
END_METHOD

METHOD RegisterMoverList : BOOL
VAR_INPUT
    NewMoverList : iMoverList;
END_VAR
(*
	Adds an entire MoverList to the Tracked Movers of the objective.
*)

PositionTrigger.RegisterMoverList(NewMoverList);
END_METHOD

{attribute 'monitoring' := 'call'}
PROPERTY TrackedMoverCount : USINT
GET
VAR
    i : INT;
END_VAR
internalTrackedMoverCount	:= 0;
FOR i := 0 TO GVL.MULTISTN_NUM_STN DO
	internalTrackedMoverCount	:= internalTrackedMoverCount + Station[i].TrackedMoverCount;
END_FOR
TrackedMoverCount	:= internalTrackedMoverCount;
END_GET
END_PROPERTY

PROPERTY TrackId : DINT
GET
TrackId := internalTrackId;
END_GET
SET
internalTrackId := TrackId;
END_SET
END_PROPERTY

METHOD UnregisterAll : BOOL
// Blow out the tracked mover array
PositionTrigger.UnregisterAll();
FOR i := 0 TO GVL.MULTISTN_NUM_STN - 1 DO
	Station[i].UnregisterAll();
END_FOR
END_METHOD

METHOD UnregisterCurrent : BOOL
VAR_INPUT
END_VAR
PositionTrigger.UnregisterCurrent();
END_METHOD

METHOD UnregisterMover : BOOL
VAR_INPUT
    RemovingMover : REFERENCE TO Mover;
END_VAR
PositionTrigger.UnregisterMover(RemovingMover);
END_METHOD

END_FUNCTION_BLOCK

// ---- POUs/XTS/BallPrinterStations/PrintStation.TcPOU
FUNCTION_BLOCK PrintStation EXTENDS MachineStation
VAR_INPUT
	rIO				: REFERENCE TO Print_IO_typ;
	rMultiStn		: REFERENCE TO MultiStation;
	rVisionStation	: REFERENCE TO Station;
	rKickoutStation	: REFERENCE TO Station;
	NumIndex		: USINT;
	NumColor		: USINT;
END_VAR
VAR_OUTPUT
END_VAR
VAR
	PosTriggerPayload	: Payload_typ;
	StationPayload		: ARRAY[0..GVL.MULTISTN_NUM_STN - 1] OF Payload_typ;
	MoverHalted			: BOOL;
	PrintConfig			: PrintConfig_typ;
	i					: INT;
	FarthestIndex0StnTrackedMovers: INT;
END_VAR

IF NOT (__ISVALIDREF(rMultiStn) AND __ISVALIDREF(rIO) AND __ISVALIDREF(rVisionStation) AND __ISVALIDREF(rKickoutStation)) THEN
	ADSLOGSTR( ADSLOG_MSGTYPE_ERROR, 'Invalid reference at %s.', InstancePath);	// how to make this work?
	RETURN;
END_IF

// Station Sequence
IF Enable THEN
	IF NOT _Enable THEN
		ACT_ConfigurePrint();
	END_IF

	// Catch Incoming Shuttles and process them
	IF rMultiStn.PositionTrigger.MoverPassedPosition THEN
(*		PosTriggerPayload	:= rMultiStn.PositionTrigger.CurrentMover.Payload;
		// Mover payload not valid for printing
		IF PosTriggerPayload.Reject OR NOT(PosTriggerPayload.HasBall AND PosTriggerPayload.BallSeated) THEN		
			PosTriggerPayload.Reject	:= TRUE;
			IF rMultiStn.TrackedMoverCount > 0 THEN
				MoverHalted				:= TRUE;
				rMultiStn.PositionTrigger.CurrentMover.Halt();
			ELSE
				rMultiStn.PositionTrigger.CurrentMover.MoveToStation(rKickoutStation);
				rMultiStn.PositionTrigger.CurrentMover.Payload	:= PosTriggerPayload;
				rMultiStn.PositionTrigger.MuteCurrent();
				MoverHalted				:= FALSE;
			END_IF
		// mover ok to print
		ELSE						*) // This doesn't work and it's not really necessary.  
										// PositionTrigger would need to buffer events.  
										// this only works when movers are going slow
										// Peter eventually going to add event buffering to position trigger, not worth doing for demo
			FarthestIndex0StnTrackedMovers	:= 100;
			FOR i := PrintConfig.LastProcessIndex0StnIndex TO 0 BY -1 DO
				IF rMultiStn.Station[i].TrackedMoverCount < FarthestIndex0StnTrackedMovers THEN
					FarthestIndex0StnTrackedMovers	:= i;
				END_IF
			END_FOR
					
			FOR i := PrintConfig.LastProcessIndex0StnIndex TO 0 BY -1 DO
				IF PrintConfig.StationEnable[i] AND PrintConfig.ProcessIndex[i] = 0 AND rMultiStn.Station[i].TrackedMoverCount = 0 THEN
					rMultiStn.PositionTrigger.CurrentMover.MoveToStation(rMultiStn.Station[i]);
					rMultiStn.PositionTrigger.MuteCurrent();
					EXIT;
				ELSIF i = 0 THEN
					rMultiStn.PositionTrigger.CurrentMover.MoveToStation(rMultiStn.Station[FarthestIndex0StnTrackedMovers]);
					rMultiStn.PositionTrigger.MuteCurrent();
					EXIT;
				END_IF
			END_FOR
		(*END_IF*)
	END_IF

	// Printing Sequence State Machine
	CASE State OF
		STN_WAIT:
			IF Run AND_THEN THIS^.MoversReadyForCycle() THEN
				FOR i := 0 TO GVL.MULTISTN_NUM_STN - 1 DO
					IF rMultiStn.Station[i].TrackedMoverCount > 0 THEN
						StationPayload[i]	:= rMultiStn.Station[i].CurrentMover.Payload;
					END_IF
				END_FOR
				rIO.Outputs.Print	:= TRUE;
				State				:= STN_PROCESS;
			END_IF

		STN_PROCESS:
			IF rIO.Inputs.PrintComplete THEN
				rIO.Outputs.Print		:= FALSE;
				FOR i := 0 TO GVL.MULTISTN_NUM_STN - 1 DO
					IF rMultiStn.Station[i].TrackedMoverCount > 0 THEN
						StationPayload[i].PrintStepComplete[PrintConfig.ProcessIndex[i]]	:= TRUE;
						IF PrintConfig.FinalPrint[i] THEN StationPayload[i].PrintComplete		:= TRUE; END_IF
					END_IF
				END_FOR
			State	:= STN_SEND;
			END_IF

		STN_SEND:

			// Write Payload Data
			FOR i := 0 TO GVL.MULTISTN_NUM_STN - 1 DO
				IF rMultiStn.Station[i].TrackedMoverCount > 0 THEN
					rMultiStn.Station[i].CurrentMover.Payload							:= StationPayload[i];
				END_IF
			END_FOR

			// Send Mover
			ACT_PrintSendMover();
			State	:= STN_WAIT;

		STN_ERROR:

	END_CASE

ELSIF _Enable THEN
	State	:= STN_WAIT;
END_IF

//Save Previous Values
_Enable	:= Enable;

ACTION ACT_ConfigurePrint:
memset(ADR(PrintConfig), 0, SIZEOF(PrintConfig));

CASE NumColor OF
1:
	CASE NumIndex OF
	1:	PrintConfig.StationEnable[2] := TRUE;	PrintConfig.ProcessIndex[2] := 0; PrintConfig.FinalPrint[2] := TRUE;	PrintConfig.LastProcessIndex0StnIndex	:= 2;

	2:	PrintConfig.StationEnable[1] := TRUE;	PrintConfig.ProcessIndex[1] := 0; PrintConfig.FinalPrint[1] := TRUE;
		PrintConfig.StationEnable[2] := TRUE;	PrintConfig.ProcessIndex[2] := 0; PrintConfig.FinalPrint[2] := TRUE;	PrintConfig.LastProcessIndex0StnIndex	:= 2;

	3:	PrintConfig.StationEnable[1] := TRUE;	PrintConfig.ProcessIndex[1] := 0; PrintConfig.FinalPrint[1] := TRUE;
		PrintConfig.StationEnable[2] := TRUE;	PrintConfig.ProcessIndex[2] := 0; PrintConfig.FinalPrint[2] := TRUE;
		PrintConfig.StationEnable[3] := TRUE;	PrintConfig.ProcessIndex[3] := 0; PrintConfig.FinalPrint[3] := TRUE;	PrintConfig.LastProcessIndex0StnIndex	:= 3;

	4:	PrintConfig.StationEnable[0] := TRUE;	PrintConfig.ProcessIndex[0] := 0; PrintConfig.FinalPrint[0] := TRUE;
		PrintConfig.StationEnable[1] := TRUE;	PrintConfig.ProcessIndex[1] := 0; PrintConfig.FinalPrint[1] := TRUE;
		PrintConfig.StationEnable[2] := TRUE;	PrintConfig.ProcessIndex[2] := 0; PrintConfig.FinalPrint[2] := TRUE;
		PrintConfig.StationEnable[3] := TRUE;	PrintConfig.ProcessIndex[3] := 0; PrintConfig.FinalPrint[3] := TRUE;	PrintConfig.LastProcessIndex0StnIndex	:= 3;
	END_CASE
2:
	CASE NumIndex OF
	1:	PrintConfig.StationEnable[1] := TRUE;	PrintConfig.ProcessIndex[1] := 0; PrintConfig.FinalPrint[1] := FALSE;	PrintConfig.LastProcessIndex0StnIndex	:= 1;
		PrintConfig.StationEnable[2] := TRUE;	PrintConfig.ProcessIndex[2] := 1; PrintConfig.FinalPrint[2] := TRUE;

	2:	PrintConfig.StationEnable[0] := TRUE;	PrintConfig.ProcessIndex[0] := 0; PrintConfig.FinalPrint[0] := FALSE;
		PrintConfig.StationEnable[1] := TRUE;	PrintConfig.ProcessIndex[1] := 0; PrintConfig.FinalPrint[1] := FALSE;	PrintConfig.LastProcessIndex0StnIndex	:= 1;
		PrintConfig.StationEnable[2] := TRUE;	PrintConfig.ProcessIndex[2] := 1; PrintConfig.FinalPrint[2] := TRUE;
		PrintConfig.StationEnable[3] := TRUE;	PrintConfig.ProcessIndex[3] := 1; PrintConfig.FinalPrint[3] := TRUE;
	END_CASE
3:
		PrintConfig.StationEnable[1] := TRUE;	PrintConfig.ProcessIndex[1] := 0; PrintConfig.FinalPrint[1] := FALSE;	PrintConfig.LastProcessIndex0StnIndex	:= 1;
		PrintConfig.StationEnable[2] := TRUE;	PrintConfig.ProcessIndex[2] := 1; PrintConfig.FinalPrint[2] := FALSE;
		PrintConfig.StationEnable[3] := TRUE;	PrintConfig.ProcessIndex[3] := 2; PrintConfig.FinalPrint[3] := TRUE;

4:		PrintConfig.StationEnable[0] := TRUE;	PrintConfig.ProcessIndex[0] := 0; PrintConfig.FinalPrint[0] := FALSE;	PrintConfig.LastProcessIndex0StnIndex	:= 0;
		PrintConfig.StationEnable[1] := TRUE;	PrintConfig.ProcessIndex[1] := 1; PrintConfig.FinalPrint[1] := FALSE;
		PrintConfig.StationEnable[2] := TRUE;	PrintConfig.ProcessIndex[2] := 2; PrintConfig.FinalPrint[2] := FALSE;
		PrintConfig.StationEnable[3] := TRUE;	PrintConfig.ProcessIndex[3] := 3; PrintConfig.FinalPrint[3] := TRUE;
END_CASE
END_ACTION

ACTION ACT_PrintSendMover:
CASE NumColor OF
1:
	CASE NumIndex OF
	1:	IF rMultiStn.Station[2].TrackedMoverCount > 0 THEN rMultiStn.Station[2].CurrentMover.MoveToStation(rVisionStation);			rMultiStn.Station[2].UnregisterCurrent();	END_IF

	2:	IF rMultiStn.Station[2].TrackedMoverCount > 0 THEN rMultiStn.Station[2].CurrentMover.MoveToStation(rVisionStation);			rMultiStn.Station[2].UnregisterCurrent();	END_IF
		IF rMultiStn.Station[1].TrackedMoverCount > 0 THEN rMultiStn.Station[1].CurrentMover.MoveToStation(rVisionStation);			rMultiStn.Station[1].UnregisterCurrent();	END_IF

	3:	IF rMultiStn.Station[3].TrackedMoverCount > 0 THEN rMultiStn.Station[3].CurrentMover.MoveToStation(rVisionStation);			rMultiStn.Station[3].UnregisterCurrent();	END_IF
		IF rMultiStn.Station[2].TrackedMoverCount > 0 THEN rMultiStn.Station[2].CurrentMover.MoveToStation(rVisionStation);			rMultiStn.Station[2].UnregisterCurrent();	END_IF
		IF rMultiStn.Station[1].TrackedMoverCount > 0 THEN rMultiStn.Station[1].CurrentMover.MoveToStation(rVisionStation);			rMultiStn.Station[1].UnregisterCurrent();	END_IF

	4:	IF rMultiStn.Station[3].TrackedMoverCount > 0 THEN rMultiStn.Station[3].CurrentMover.MoveToStation(rVisionStation);			rMultiStn.Station[3].UnregisterCurrent();	END_IF
		IF rMultiStn.Station[2].TrackedMoverCount > 0 THEN rMultiStn.Station[2].CurrentMover.MoveToStation(rVisionStation);			rMultiStn.Station[2].UnregisterCurrent();	END_IF
		IF rMultiStn.Station[1].TrackedMoverCount > 0 THEN rMultiStn.Station[1].CurrentMover.MoveToStation(rVisionStation);			rMultiStn.Station[1].UnregisterCurrent();	END_IF
		IF rMultiStn.Station[0].TrackedMoverCount > 0 THEN rMultiStn.Station[0].CurrentMover.MoveToStation(rVisionStation);			rMultiStn.Station[0].UnregisterCurrent();	END_IF
	END_CASE
2:
	CASE NumIndex OF
	1:	IF rMultiStn.Station[2].TrackedMoverCount > 0 THEN rMultiStn.Station[2].CurrentMover.MoveToStation(rVisionStation);			rMultiStn.Station[2].UnregisterCurrent();	END_IF
		IF rMultiStn.Station[1].TrackedMoverCount > 0 THEN rMultiStn.Station[1].CurrentMover.MoveToStation(rMultiStn.Station[2]);	rMultiStn.Station[1].UnregisterCurrent();	END_IF


	2:	IF rMultiStn.Station[3].TrackedMoverCount > 0 THEN rMultiStn.Station[3].CurrentMover.MoveToStation(rVisionStation);			rMultiStn.Station[3].UnregisterCurrent();	END_IF
		IF rMultiStn.Station[2].TrackedMoverCount > 0 THEN rMultiStn.Station[2].CurrentMover.MoveToStation(rVisionStation);			rMultiStn.Station[2].UnregisterCurrent();	END_IF
		IF rMultiStn.Station[1].TrackedMoverCount > 0 THEN rMultiStn.Station[1].CurrentMover.MoveToStation(rMultiStn.Station[3]);	rMultiStn.Station[1].UnregisterCurrent();	END_IF
		IF rMultiStn.Station[0].TrackedMoverCount > 0 THEN rMultiStn.Station[0].CurrentMover.MoveToStation(rMultiStn.Station[2]);	rMultiStn.Station[0].UnregisterCurrent();	END_IF
	END_CASE

3:		IF rMultiStn.Station[3].TrackedMoverCount > 0 THEN rMultiStn.Station[3].CurrentMover.MoveToStation(rVisionStation);			rMultiStn.Station[3].UnregisterCurrent();	END_IF
		IF rMultiStn.Station[2].TrackedMoverCount > 0 THEN rMultiStn.Station[2].CurrentMover.MoveToStation(rMultiStn.Station[3]);	rMultiStn.Station[2].UnregisterCurrent();	END_IF
		IF rMultiStn.Station[1].TrackedMoverCount > 0 THEN rMultiStn.Station[1].CurrentMover.MoveToStation(rMultiStn.Station[2]);	rMultiStn.Station[1].UnregisterCurrent();	END_IF

4:		IF rMultiStn.Station[3].TrackedMoverCount > 0 THEN rMultiStn.Station[3].CurrentMover.MoveToStation(rVisionStation);			rMultiStn.Station[3].UnregisterCurrent();	END_IF
		IF rMultiStn.Station[2].TrackedMoverCount > 0 THEN rMultiStn.Station[2].CurrentMover.MoveToStation(rMultiStn.Station[3]);	rMultiStn.Station[2].UnregisterCurrent();	END_IF
		IF rMultiStn.Station[1].TrackedMoverCount > 0 THEN rMultiStn.Station[1].CurrentMover.MoveToStation(rMultiStn.Station[2]);	rMultiStn.Station[1].UnregisterCurrent();	END_IF
		IF rMultiStn.Station[0].TrackedMoverCount > 0 THEN rMultiStn.Station[0].CurrentMover.MoveToStation(rMultiStn.Station[1]);	rMultiStn.Station[0].UnregisterCurrent();	END_IF
END_CASE
END_ACTION

ACTION ACT_PrintStatuses:

END_ACTION

METHOD MoversReadyForCycle : BOOL
// Check that all movers are in position, and that there are movers in all of the enabled process index 0 print positions
MoversReadyForCycle	:= TRUE; 
IF NOT rMultiStn.AllMoversInPosition THEN	// Any stations with tracked movers that don't have mover in position will trigger this false
	MoversReadyForCycle	:= FALSE;
ELSE
	FOR i := GVL.MULTISTN_NUM_STN - 1 TO 0 BY - 1 DO
		IF PrintConfig.StationEnable[i] AND PrintConfig.ProcessIndex[i] = 0 THEN	// Check that all process index 0 stations have movers to ensure full print cycle
			IF rMultiStn.Station[i].TrackedMoverCount = 0 AND NOT MoverHalted THEN		// Ignore this check if there is a mover halted by the position trigger
				MoversReadyForCycle	:= FALSE;
			END_IF
		END_IF
	END_FOR
END_IF
END_METHOD

END_FUNCTION_BLOCK

// ---- POUs/XTS/Zone.TcPOU
{attribute 'hide_all_local'}
FUNCTION_BLOCK Zone EXTENDS Objective
VAR

    internalStartPosition	: LREAL;
    internalEndPosition  	: LREAL;
    internalDirection    	: Tc2_MC2.MC_Direction;
	internalTrackId			: DINT := 1;

    internalMoverList : MoverList;

END_VAR

PROPERTY CurrentMoverList : iMoverList
GET
VAR
    i : ulint;
	moverTrackId: INT;
END_VAR
internalMoverList.UnregisterAll();

FOR i := 0 TO SIZEOF(TrackedMovers) / SIZEOF(internalTrackedMovers[0]) - 1 DO
    IF internalTrackedMovers[i] <> 0 THEN
		moverTrackId := internalTrackedMovers[i]^.CurrentTrack^.Id;
		IF (moverTrackId = internalTrackId) THEN
			IF internalStartPosition < internalEndPosition
				   AND internalTrackedMovers[i]^.TrackInfo.TrackPosition > internalStartPosition
				   AND internalTrackedMovers[i]^.TrackInfo.TrackPosition < internalEndPosition THEN
				// Zone does NOT contain the rollover point, and DOES contain the mover
	
				internalMoverList.RegisterMover(internalTrackedMovers[i]^);
	
			ELSIF internalStartPosition > internalEndPosition
					  AND (internalTrackedMovers[i]^.TrackInfo.TrackPosition > internalStartPosition
					  OR internalTrackedMovers[i]^.TrackInfo.TrackPosition < internalEndPosition) THEN
				// Zone DOES contain the rollover point, and DOES contain the mover
	
				internalMoverList.RegisterMover(internalTrackedMovers[i]^);
	
			ELSE
				// Either the zone doesn't contain this mover,
				// Or the StartPosition and EndPosition are coincident. Either way, add no movers
			END_IF
		END_IF
    END_IF
END_FOR

CurrentMoverList := internalMoverList;
END_GET
END_PROPERTY

PROPERTY EndPosition : LREAL
GET
EndPosition := internalEndPosition;
END_GET
SET
// todo add limit checks?
internalEndPosition := EndPosition;
END_SET
END_PROPERTY

METHOD GetMover : REFERENCE TO Mover
VAR_INPUT
    Index     : USINT;                // 0 is find the first closest mover, 1 is find the second closest mover, 2 is find the third, etc. etc. etc.
    Direction : Tc2_MC2.MC_Direction; // Positive = find the mover closest to the End Position. Negative = find the mover closest to the Start Position
END_VAR



IF Direction = MC_Positive_Direction THEN
    GetMover REF= THIS^.CurrentMoverList.GetMoverByLocation(Index, THIS^.EndPosition, MC_Positive_Direction);
	GetMover.SourceInstancePath		:= THIS^.InstancePath;
ELSIF Direction = MC_Negative_Direction THEN
    GetMover REF= THIS^.CurrentMoverList.GetMoverByLocation(Index, THIS^.StartPosition, MC_Negative_Direction);
	GetMover.SourceInstancePath		:= THIS^.InstancePath;
ELSE
    GetMover REF= 0;
END_IF

// If the Zone has no mover to return given the input parameters, then return an imposter ErrorMover
IF __ISVALIDREF(GetMover) = FALSE THEN
	ErrorMover.SourceInstancePath	:= THIS^.InstancePath;
	GetMover						REF= ErrorMover;
END_IF
END_METHOD

PROPERTY StartPosition : LREAL
GET
StartPosition := internalStartPosition;
END_GET
SET
// Todo add limit checks?
internalStartPosition := StartPosition;
END_SET
END_PROPERTY

PROPERTY TrackId : DINT
GET
TrackId := internalTrackId;
END_GET
SET
internalTrackId := TrackId;
END_SET
END_PROPERTY

{attribute 'monitoring' := 'call'}
PROPERTY ZoneLength : LREAL
GET
IF internalStartPosition < internalEndPosition THEN
    // Zone does NOT include the rollover point
    ZoneLength := internalEndPosition - internalStartPosition;
ELSIF internalStartPosition > internalEndPosition THEN
    // Zone DOES include the rollover point
    ZoneLength := internalEndPosition + (internalEndPosition + GVL.TRACK_LENGTH - internalStartPosition);
ELSE
    // Start and end position are coincident, ZL is 0
    ZoneLength := 0;
END_IF
END_GET
END_PROPERTY

END_FUNCTION_BLOCK

// ---- VISUs/Controls.TcVIS
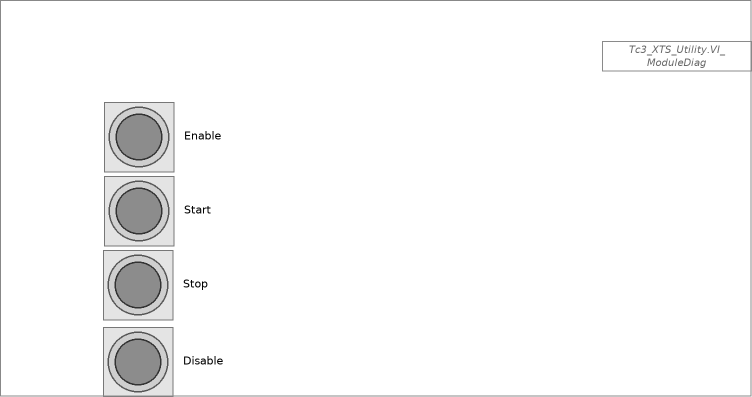
VISUALIZATION Controls  // 752x397
    PushSwitchLed (104,102 70x70), variable: MAIN.MainCommands.Enable, behaviour: TOGGLE, style: Switch-PushSwitchLed-Gray
    Label (181,121 150x30), "Enable"
    Label (181,195 150x30), "Start"
    PushSwitchLed (104,176 70x70), variable: MAIN.MainCommands.Start, behaviour: TOGGLE, style: Switch-PushSwitchLed-Gray
    Label (180,269 150x30), "Stop"
    PushSwitchLed (103,250 70x70), variable: MAIN.MainCommands.Stop, behaviour: TOGGLE, style: Switch-PushSwitchLed-Gray
    Label (180,346 150x30), "Disable"
    PushSwitchLed (103,327 70x70), variable: MAIN.MainCommands.Disable, behaviour: TOGGLE, style: Switch-PushSwitchLed-Gray
    Frame (602,41 150x30)
        shows Tc3_XTS_Utility.VI_ModuleDiag()
END_VISUALIZATION
